FUNCTION_BLOCK C_RESTFUL_CLIENT
VAR_INPUT
END_VAR
VAR_OUTPUT
END_VAR
VAR
	_ifc_Communication 	: IFC_GENERIC_COMMUNICATION_INTERFACE;
	_c_HttpRequest		: C_HTTP_REQUEST;
END_VAR

END_FUNCTION_BLOCK

(* stored: Version 1.1.0.1, ProductVersion 3.1.4019.2
   POU C_RESTFUL_CLIENT: Id {4563b6e5-238a-4d52-b7b2-2e9aa16a0d74}, SpecialFunc None *)
